FUNCTION_BLOCK Central_Server (* Basic Function Block Type *)
  (* Standard: 61499-2 *)
  (* Version 0.2, 2003-12-04, JHC, Rockwell Automation, Renamed for better indexing. *)
  (* Version 0.1, 2002-11-05, JHC, Rockwell Automation, Corrected missing ST element in Algorithm REQ. *)
  (* Version 0.0, 2000-05-30, JHC, Rockwell Automation *)
  (* Compiler header: package fb.rt.cs725; *)
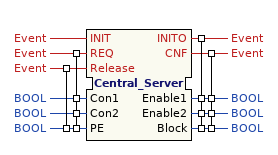
  EVENT_INPUT
    INIT; (* Initialization Request *)
    REQ WITH Con1, Con2, PE; (* Normal Execution Request *)
    Release WITH PE;
  END_EVENT
  EVENT_OUTPUT
    INITO WITH Enable1, Enable2, Block; (* Initialization Confirm *)
    CNF WITH Enable2, Enable1, Block; (* Execution Confirmation *)
  END_EVENT
  VAR_INPUT
    Con1 : BOOL;
    Con2 : BOOL;
    PE : BOOL;
  END_VAR
  VAR_OUTPUT
    Enable1 : BOOL;
    Enable2 : BOOL;
    Block : BOOL;
  END_VAR
  VAR
    queue1 : INT := 0;
    queue2 : INT := 0;
    queue3 : INT := 0;
    token : BOOL;
    Con1_prev : BOOL;
    Con2_prev : BOOL;
    PE_prev : BOOL;
  END_VAR
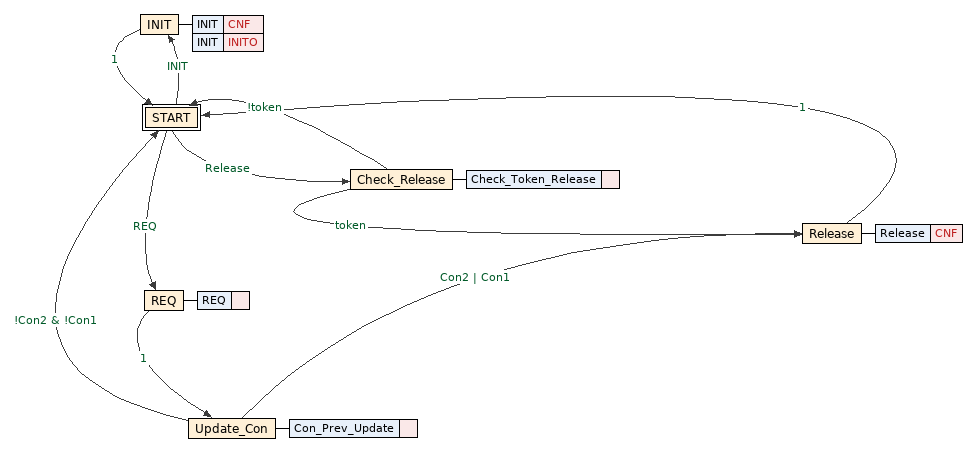
  EC_STATES
    START; (* Initial State *)
    INIT : INIT -> CNF, INIT -> INITO; (* Initialization *)
    REQ : REQ; (* Normal execution *)
    Release : Release -> CNF;
    Check_Release : Check_Token_Release;
    Update_Con : Con_Prev_Update;
  END_STATES
  EC_TRANSITIONS
    START TO INIT := INIT;
    INIT TO START := 1;
    Release TO START := 1;
    START TO Check_Release := Release;
    Check_Release TO Release := token;
    START TO REQ := REQ;
    Check_Release TO START := !token;
    REQ TO Update_Con := 1;
    Update_Con TO Release := Con2 | Con1;
    Update_Con TO START := !Con2 & !Con1;
  END_TRANSITIONS
  ALGORITHM INIT IN Java: (* Initialization algorithm *)
Enable1.value=false;
Enable2.value=false;
token.value=true;
Con1_prev.value=true;
Con2_prev.value=true;
  END_ALGORITHM
  ALGORITHM REQ IN Java: (* Normally executed algorithm *)
System.out.println("Request to server");
System.out.print("Conveyor 1 input status:");
System.out.println(Con1.value);
System.out.print("Conveyor 2 input status:");
System.out.println(Con2.value);

System.out.print("Conveyor 1 output status:");
System.out.println(Enable1.value);
System.out.print("Conveyor 2 output status:");
System.out.println(Enable2.value);
if (Con1.value && Con1.value != Con1_prev.value){
if (queue1.value == 0){
queue1.value=1;
}else if (queue2.value == 0){
queue2.value=1;
}else{
queue3.value=1;
}
Enable1.value=true;
}
if (Con2.value && Con2.value != Con2_prev.value){
if (queue1.value == 0){
queue1.value=2;
}else if (queue2.value == 0){
queue2.value=2;
}else{
queue3.value=2;
}
Enable2.value=true;
}
  END_ALGORITHM
  ALGORITHM Release IN Java:
System.out.println("QUEUE:");
System.out.println(queue1);
System.out.println(queue2);
System.out.println(queue3);

System.out.print("RELEASE SENSOR:");
System.out.println(PE.value);

if(token.value){
if(queue1.value!=0){
if(queue1.value==1){
Enable1.value=false;
System.out.print("Input 1 has accessed section");
}else{
Enable2.value=false;
System.out.print("Input 2 has accessed section");
}
token.value=false;
queue1.value=queue2.value;
queue2.value=queue3.value;
queue3.value=0;
}else{
Enable1.value=false;
Enable2.value=false;
}
}
  END_ALGORITHM
  ALGORITHM Check_Token_Release IN Java:
if(PE_prev.value != PE.value){
if(PE.value == false){
token.value=true;
}
PE_prev.value=PE.value;
}
  END_ALGORITHM
  ALGORITHM Con_Prev_Update IN Java:
Con1_prev.value=Con1.value;
Con2_prev.value=Con2.value;
  END_ALGORITHM
END_FUNCTION_BLOCK
